// Mitsubishi GX Works2 project: 2026_01_21_PASSIVITY_AUTO   PLC: Q03UDV

PROGRAM MAIN
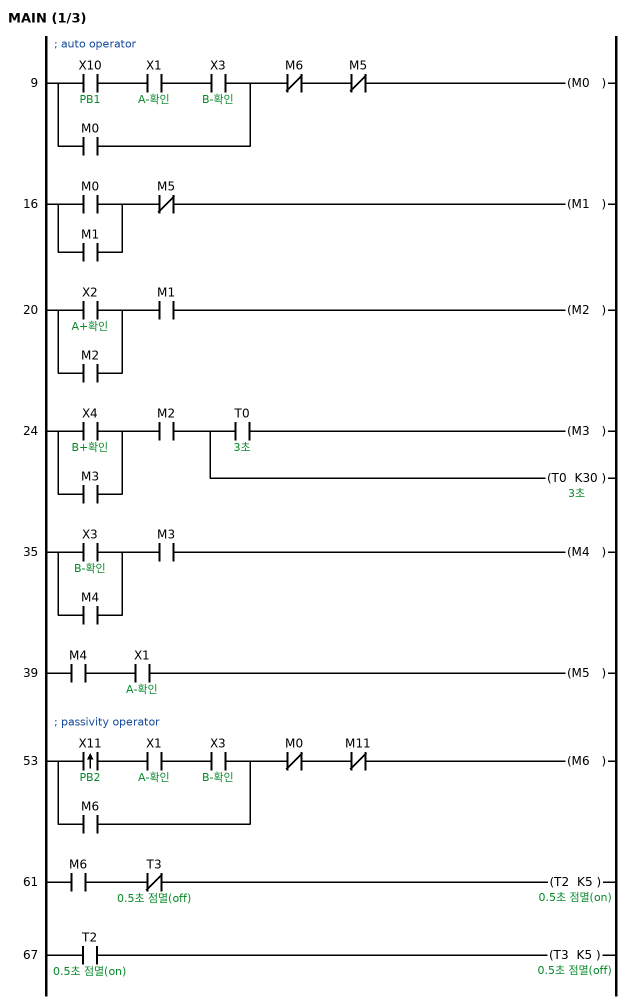
; auto operator
9     LD      X10  ; PB1
      AND     X1  ; A-확인
      AND     X3  ; B-확인
      OR      M0
      ANI     M6
      ANI     M5
      OUT     M0
16    LD      M0
      OR      M1
      ANI     M5
      OUT     M1
20    LD      X2  ; A+확인
      OR      M2
      AND     M1
      OUT     M2
24    LD      X4  ; B+확인
      OR      M3
      AND     M2
      MPS
      AND     T0  ; 3초
      OUT     M3
      MPP
      OUT     T0 K30  ; 3초
35    LD      X3  ; B-확인
      OR      M4
      AND     M3
      OUT     M4
39    LD      M4
      AND     X1  ; A-확인
      OUT     M5
; passivity operator
53    LDP     X11  ; PB2
      AND     X1  ; A-확인
      AND     X3  ; B-확인
      OR      M6
      ANI     M0
      ANI     M11
      OUT     M6
61    LD      M6
      ANI     T3  ; 0.5초 점멸(off)
      OUT     T2 K5  ; 0.5초 점멸(on)
67    LD      T2  ; 0.5초 점멸(on)
      OUT     T3 K5  ; 0.5초 점멸(off)
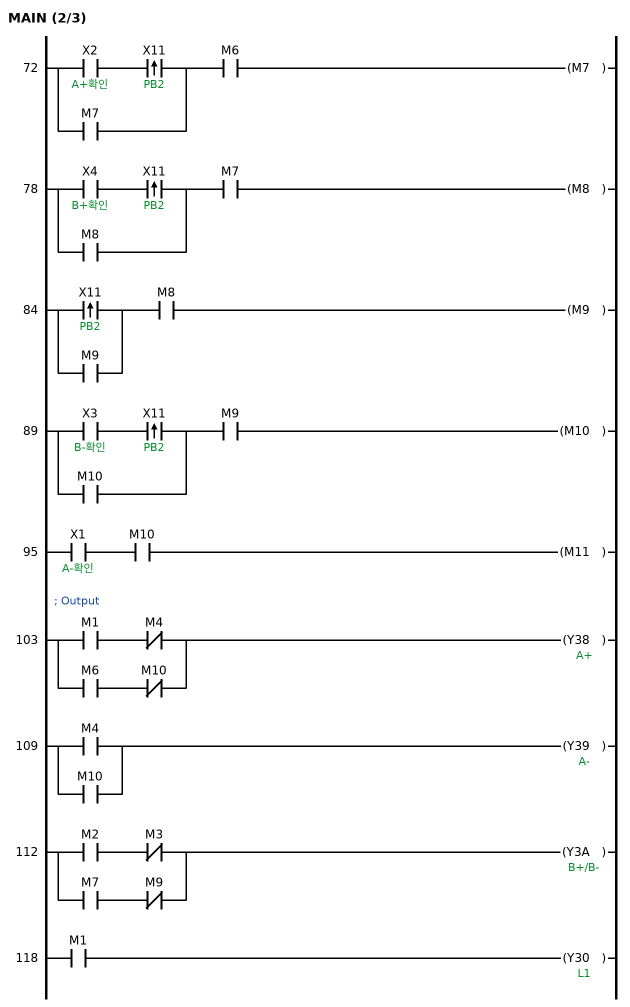
72    LD      X2  ; A+확인
      ANDP    X11  ; PB2
      OR      M7
      AND     M6
      OUT     M7
78    LD      X4  ; B+확인
      ANDP    X11  ; PB2
      OR      M8
      AND     M7
      OUT     M8
84    LDP     X11  ; PB2
      OR      M9
      AND     M8
      OUT     M9
89    LD      X3  ; B-확인
      ANDP    X11  ; PB2
      OR      M10
      AND     M9
      OUT     M10
95    LD      X1  ; A-확인
      AND     M10
      OUT     M11
; Output
103   LD      M1
      ANI     M4
      LD      M6
      ANI     M10
      ORB
      OUT     Y38  ; A+
109   LD      M4
      OR      M10
      OUT     Y39  ; A-
112   LD      M2
      ANI     M3
      LD      M7
      ANI     M9
      ORB
      OUT     Y3A  ; B+/B-
118   LD      M1
      OUT     Y30  ; L1
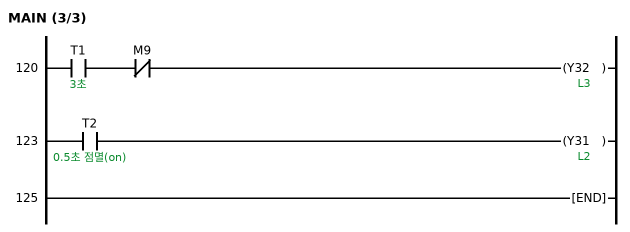
120   LD      T1  ; 3초
      ANI     M9
      OUT     Y32  ; L3
123   LD      T2  ; 0.5초 점멸(on)
      OUT     Y31  ; L2
125   END
END_PROGRAM
